FUNCTION_BLOCK "LAxisCtrlApcFr_ChangeModulo"
TITLE = Execute Template
{ S7_Optimized_Access := 'TRUE' }
AUTHOR : SDA
FAMILY : APCFR
VERSION : 1.0
//Template for an FB with Execute / Busy / Done Handling according to PLC Open "Function Blocks for Motion Control"
   VAR_INPUT
      execute { ExternalAccessible := 'False'; ExternalVisible := 'False'; ExternalWritable := 'False'} : Bool;   // Rising edge starts action once
      moduloStartValue { ExternalAccessible := 'False'; ExternalVisible := 'False'; ExternalWritable := 'False'} : LReal;
      moduloLength { ExternalAccessible := 'False'; ExternalVisible := 'False'; ExternalWritable := 'False'} : LReal := 360.0;
      axis { ExternalAccessible := 'False'; ExternalVisible := 'False'; ExternalWritable := 'False'} : DB_ANY;
   END_VAR

   VAR_OUTPUT
      done { ExternalAccessible := 'False'; ExternalVisible := 'False'; ExternalWritable := 'False'} : Bool;   // TRUE: Commanded action has been completed successfully
      busy { ExternalAccessible := 'False'; ExternalVisible := 'False'; ExternalWritable := 'False'} : Bool;   // TRUE: FB is not finished and new output values can be expected
      commandAborted { ExternalAccessible := 'False'; ExternalVisible := 'False'; ExternalWritable := 'False'} : Bool;
      error { ExternalAccessible := 'False'; ExternalVisible := 'False'; ExternalWritable := 'False'} : Bool;   // Rising edge informs that an error occurred during the execution of
      status { ExternalAccessible := 'False'; ExternalVisible := 'False'; ExternalWritable := 'False'} : Word := "STATUS_NO_CALL";   // Current status of FB
      subStatus { ExternalAccessible := 'False'; ExternalVisible := 'False'; ExternalWritable := 'False'} : Word := "ERR_NO_ERROR";
      errorValue { ExternalAccessible := 'False'; ExternalVisible := 'False'; ExternalWritable := 'False'} : Int := 0;
   END_VAR

   VAR
      statExecuteOld { ExternalAccessible := 'False'; ExternalVisible := 'False'; ExternalWritable := 'False'} : Bool;   // Old value of execute for edge detection
      statDone { ExternalAccessible := 'False'; ExternalVisible := 'False'; ExternalWritable := 'False'} : Bool;   // Static value for output done
      statBusy { ExternalAccessible := 'False'; ExternalVisible := 'False'; ExternalWritable := 'False'} : Bool;   // Static value for output busy
      statCommandAborted { ExternalAccessible := 'False'; ExternalVisible := 'False'; ExternalWritable := 'False'} : Bool;
      statError { ExternalAccessible := 'False'; ExternalVisible := 'False'; ExternalWritable := 'False'} : Bool;   // Static value for output error
      statErrorID { ExternalAccessible := 'False'; ExternalVisible := 'False'; ExternalWritable := 'False'} : Word;
      statSubErrorID { ExternalAccessible := 'False'; ExternalVisible := 'False'; ExternalWritable := 'False'} : Word;
      statErrorValue { ExternalAccessible := 'False'; ExternalVisible := 'False'; ExternalWritable := 'False'} : Int;
      statActualStep { ExternalAccessible := 'False'; ExternalVisible := 'False'; ExternalWritable := 'False'} : Int;
      statNextStep { ExternalAccessible := 'False'; ExternalVisible := 'False'; ExternalWritable := 'False'} : Int;
      InstLapcFr_WriteToParameterR_ModuloLength { ExternalAccessible := 'False'; ExternalVisible := 'False'; ExternalWritable := 'False'; S7_SetPoint := 'False'} : "LAxisCtrlApcFr_WriteToParameter";
      InstLapcFr_WriteToParameter_ModuloStartValue { ExternalAccessible := 'False'; ExternalVisible := 'False'; ExternalWritable := 'False'; S7_SetPoint := 'False'} : "LAxisCtrlApcFr_WriteToParameter";
      statStepTimeOut_IN { ExternalAccessible := 'False'; ExternalVisible := 'False'; ExternalWritable := 'False'} : Bool;
      statStepTimeOut_PT { ExternalAccessible := 'False'; ExternalVisible := 'False'; ExternalWritable := 'False'} : Time;
      instStepTimeOut {InstructionName := 'TON_TIME'; LibVersion := '1.0'; ExternalAccessible := 'False'; ExternalVisible := 'False'; ExternalWritable := 'False'; S7_SetPoint := 'False'} : TON_TIME;
   END_VAR

   VAR_TEMP
      tempRefPosAxis {InstructionName := 'TO_PositioningAxis'; LibVersion := '8.0'} : REF_TO TO_PositioningAxis;   // Temporary reference of the technology object type TO_PositioningAxis
   END_VAR


BEGIN
	REGION HEADER
	  //===================================================================================================
	  // SIEMENS SAS    RC-FR DI FA APC
	  //---------------------------------------------------------------------------------------------------
	  // Restrictions:  ---
	  // Requirements:  ---
	  //---------------------------------------------------------------------------------------------------
	  // Description:   Changing modulo value of axis
	  //---------------------------------------------------------------------------------------------------
	  // Change log table:
	  // Version  Date        TIA   Expert  Changes applied
	  // 01.00    2020.07.24  V16   SDA     First released version
	  // 01.01    2021.06.01  V16   SDA     Name changed
	  // 01.02    2022.04.20  V17   FGe     Bugfix: incorrect error value step 40
	  //                                    Moved constants TO global definition
	  // 05.00    2024.09.11  V19   SDa     Adaptation with DBAny type #axis
	  //---------------------------------------------------------------------------------------------------
	  // Compatibility to TIA version require the use of latest version for PLC fimware and Motion Control
	  // e.g; Firmware 3.1 and Motion Control V8.0 for TIA V19
	  //===========================================================================================
	END_REGION

	REGION INITIALISATION
	    #tempRefPosAxis ?= #axis;
	END_REGION

	IF (#tempRefPosAxis <> NULL) THEN
	    // Axis type is TO_PositioningAxis or TO_SynchronousAxis

	    REGION INSTANCES
	        //------------------------------------------------------------------------------------------
	        // TODO: Insert here instances of MC instructions.
	        // inputs / outputs to be set / used in main section

	        #instStepTimeOut(IN := #statStepTimeOut_IN,
	                         PT := #statStepTimeOut_PT);

	        #InstLapcFr_WriteToParameterR_ModuloLength("TO" := #tempRefPosAxis^,
	                                                   restart := false,
	                                                   parameterValue := #moduloLength,
	                                                   TO_Parameter := #tempRefPosAxis^.Modulo.Length);

	        #InstLapcFr_WriteToParameter_ModuloStartValue("TO" := #tempRefPosAxis^,
	                                                      restart := true,
	                                                      parameterValue := #moduloStartValue,
	                                                      TO_Parameter := #tempRefPosAxis^.Modulo.StartValue);
	        //-----------------------------------------------------------------------------------
	    END_REGION

	    REGION CALL HANDLING

	        //Check if FB is triggered
	        IF #execute AND NOT #statExecuteOld
	            // if FB should finish current job before new job can be started with rising edge of execute,
	            // you must remove the first comment character on next line
	            AND NOT #statBusy
	        THEN
	            REGION FB TRIG (FIRST CALL)
	                //-----------------------------------------------------------------------------------
	                //TODO: Initialize functionality after triggering FB, e.g. reset of values
	                //
	                // Timers
	                #statStepTimeOut_IN := FALSE;
	                // Commands
	                #InstLapcFr_WriteToParameterR_ModuloLength.write := FALSE;
	                #InstLapcFr_WriteToParameter_ModuloStartValue.write := FALSE;
	                // Status
	                #statNextStep := 10;
	                #statErrorID := "STATUS_FIRST_CALL";
	                #statSubErrorID := "ERR_NO_ERROR";
	                //-----------------------------------------------------------------------------------

	                //Functionality is busy
	                #statDone := FALSE;
	                #statBusy := TRUE;
	                #statCommandAborted := FALSE;
	                //Reset diagnostic
	                #statError := FALSE;
	                #statErrorID := "ERR_NO_ERROR";
	                #statSubErrorID := "ERR_NO_ERROR";
	                #statErrorValue := 0;
	                // Write outputs
	                #done := #statDone;
	                #busy := #statBusy;
	                #commandAborted := #statCommandAborted;
	                #error := #statError;
	                #status := "STATUS_FIRST_CALL";
	                #subStatus := #statSubErrorID;
	                #errorValue := #statErrorValue;
	                #statExecuteOld := #execute;
	                RETURN;
	            END_REGION

	            //FB is currently inactive
	        ELSIF NOT #execute AND NOT #statBusy AND NOT #statExecuteOld
	        THEN
	            REGION NO CALL
	                //Outputs are reset with falling edge of enable input
	                //Write outputs
	                #done := #statDone;
	                #busy := #statBusy;
	                #commandAborted := #statCommandAborted;
	                #error := #statError;
	                #status := "STATUS_NO_CALL";
	                #subStatus := "ERR_NO_ERROR";
	                #errorValue := 0;
	                #statExecuteOld := #execute;
	                RETURN;
	            END_REGION

	            //FB is currently executed and not finished
	        ELSIF #statBusy OR #execute
	        THEN
	            REGION BUSY
	                #statExecuteOld := #execute OR #statBusy;
	            END_REGION

	            //FB finished job
	        ELSE
	            REGION LAST CALL
	                //-----------------------------------------------------------------------------------
	                //TODO: Initialize functionality after triggering FB, e.g. reset of values
	                //
	                // Timers
	                #statStepTimeOut_IN := FALSE;
	                // Commands
	                #InstLapcFr_WriteToParameterR_ModuloLength.write := FALSE;
	                #InstLapcFr_WriteToParameter_ModuloStartValue.write := FALSE;
	                // State
	                #statNextStep := 0;
	                //-----------------------------------------------------------------------------------
	                #statDone := FALSE;
	                #statBusy := FALSE;
	                #statCommandAborted := FALSE;
	                #statError := FALSE;
	                #statErrorID := "ERR_NO_ERROR";
	                #statSubErrorID := "ERR_NO_ERROR";
	                #statErrorValue := 0;
	                #statExecuteOld := #execute;
	                RETURN;
	            END_REGION

	        END_IF;
	    END_REGION ;

	    REGION USER PROGRAM
	        //-----------------------------------------------------------------------------------
	        //TODO: Add user program
	        //
	        //Following values have to be set in user program:
	        //  - statDone:     FB is finished with execution
	        //  - statAborted   Execution is aborted by an external command
	        //  - statError:    Error happened in program
	        //  - statStatus:   Identifier for current error
	        //  - statSubStatus:Identifier for subcall error
	        //
	        //Following values are not allowed to use in user program:
	        //  - statBusy
	        //  - status, subStatus, aborted, busy, done and error
	        //
	        //Attention:
	        //  - Input parameters can be updated continously
	        //  - If inputs exceed application limits, system has either to throw an error or to correct it
	        //      automatically
	        //-----------------------------------------------------------------------------------

	        REGION CHANGE MODULO VALUES

	            // update running step
	            #statActualStep := #statNextStep;
	            CASE #statActualStep OF

	                10: // Init values
	                    REGION INITIALISATION
	                        // Next step
	                        #statNextStep := 20;
	                    END_REGION

	                20: // Check change modulo conditions
	                    REGION CHECK CONDITIONS
	                        IF NOT #tempRefPosAxis^.Modulo.Enable THEN
	                            // module not activated
	                            #statErrorID := "ERR_CM_MODULO_NOT_ACTIVATED";
	                            #statNextStep := 900;

	                        ELSIF #moduloLength <= 0 THEN
	                            // wrong length
	                            #statErrorID := "ERR_CM_LENGTH_VALUE";
	                            #statNextStep := 900;

	                        ELSIF #tempRefPosAxis^.StatusWord.%X0 THEN
	                            // axis enabled
	                            #statErrorID := "ERR_CM_AXIS_ENABLED";
	                            #statNextStep := 900;

	                        ELSE
	                            // Next step
	                            #statNextStep := 30;
	                        END_IF;
	                    END_REGION

	                30: // change length value
	                    REGION CHANGE MODULO LENGTH VALUE
	                        // Step timeout
	                        #statStepTimeOut_PT := "LAPCFR_CM_WRITE_TOPARAMETER_TIMEOUT";
	                        #statStepTimeOut_IN := true;

	                        #InstLapcFr_WriteToParameterR_ModuloLength.write := TRUE;

	                        IF #InstLapcFr_WriteToParameterR_ModuloLength.error THEN
	                            #statErrorID := "ERR_CM_WRITEPARAMETER_LENGTHVALUE";
	                            #statSubErrorID := #InstLapcFr_WriteToParameterR_ModuloLength.status;
	                            #InstLapcFr_WriteToParameterR_ModuloLength.write := FALSE;
	                            #statStepTimeOut_IN := FALSE;
	                            #statNextStep := 900;

	                        ELSIF #InstLapcFr_WriteToParameterR_ModuloLength.done THEN
	                            #InstLapcFr_WriteToParameterR_ModuloLength.write := FALSE;
	                            #statStepTimeOut_IN := FALSE;
	                            // Next step
	                            #statNextStep := 40;

	                        ELSIF #instStepTimeOut.Q THEN
	                            // write parameter timeout
	                            #statErrorID := "ERR_CM_WRITEPARAMETER_TIMEOUT_LENGTHVALUE";
	                            #InstLapcFr_WriteToParameterR_ModuloLength.write := FALSE;
	                            #statStepTimeOut_IN := FALSE;
	                            #statNextStep := 900;
	                        END_IF;

	                    END_REGION

	                40: // change start value
	                    REGION CHANGE MODULO START VALUE
	                        // Step timeout
	                        #statStepTimeOut_PT := "LAPCFR_CM_WRITE_TOPARAMETER_TIMEOUT";
	                        #statStepTimeOut_IN := true;

	                        #InstLapcFr_WriteToParameter_ModuloStartValue.write := TRUE;

	                        IF #InstLapcFr_WriteToParameter_ModuloStartValue.error THEN
	                            #statErrorID := "ERR_CM_WRITEPARAMETER_STARTVALUE";
	                            #statSubErrorID := #InstLapcFr_WriteToParameter_ModuloStartValue.status;
	                            #InstLapcFr_WriteToParameter_ModuloStartValue.write := FALSE;
	                            #statStepTimeOut_IN := FALSE;
	                            #statNextStep := 900;

	                        ELSIF #InstLapcFr_WriteToParameter_ModuloStartValue.done THEN
	                            #InstLapcFr_WriteToParameter_ModuloStartValue.write := FALSE;
	                            #statStepTimeOut_IN := FALSE;
	                            // Next step
	                            #statNextStep := 120;

	                        ELSIF #instStepTimeOut.Q THEN
	                            // write parameter timeout
	                            #statErrorID := "ERR_CM_WRITEPARAMETER_TIMEOUT_STARTVALUE";
	                            #InstLapcFr_WriteToParameterR_ModuloLength.write := FALSE;
	                            #InstLapcFr_WriteToParameter_ModuloStartValue.write := FALSE;
	                            #statStepTimeOut_IN := FALSE;
	                            #statNextStep := 900;
	                        END_IF;

	                    END_REGION

	                120://Function Ok
	                    REGION FUNCTION_DONE
	                        #statDone := TRUE;
	                    END_REGION ;

	                900:  //Fault handling
	                    REGION FUNCTION_FAULTY
	                        #statNextStep := 910;
	                    END_REGION

	                910:   // change modulo values ended with fault
	                    #statError := TRUE;

	            END_CASE;

	            IF #statNextStep = 900 AND #statActualStep <> 900 THEN
	                // Store faulty step
	                #statErrorValue := #statActualStep;
	            END_IF;

	        END_REGION

	        //
	        //-----------------------------------------------------------------------------------
	    END_REGION

	    REGION ERROR_HANDLING

	        //Error occured in request
	        IF #statError
	        THEN
	            #statDone := FALSE;
	            #statCommandAborted := FALSE;
	            #statBusy := FALSE;
	            //-----------------------------------------------------------------------------------
	            //TODO: Set correct status that identifies error clearly if not set in user program region
	            // #statStatus := ...;
	            // #statSubStatus := ...;
	            //
	            #status := #statErrorID;
	            #subStatus := #statSubErrorID;
	            #errorValue := #statErrorValue;
	            //-----------------------------------------------------------------------------------

	            // Resquest aborted
	        ELSIF #statCommandAborted
	        THEN
	            #statDone := FALSE;
	            #statBusy := FALSE;
	            #statError := FALSE;
	            #status := "STATUS_EXECUTION_ABORTED";
	            #subStatus := "ERR_NO_ERROR";
	            #errorValue := 0;

	            //Request finished
	        ELSIF #statDone
	        THEN
	            #statBusy := FALSE;
	            #statCommandAborted := FALSE;
	            #statError := FALSE;
	            #status := "STATUS_FINISHED_NOERROR";
	            #subStatus := "ERR_NO_ERROR";
	            #errorValue := 0;

	            //Request in execution
	        ELSE
	            #status := "STATUS_SUBSEQUENT_CALL";
	            #subStatus := "ERR_NO_ERROR";
	            #errorValue := 0;
	        END_IF;

	        //Write static values to outputs
	        #done := #statDone;
	        #busy := #statBusy;
	        #commandAborted := #statCommandAborted;
	        #error := #statError;
	    END_REGION
	    //-----------------------------------------------------------------------------------

	ELSE
	    IF #execute THEN
	        // Invalid TO specification
	        #error := TRUE;
	        #done := FALSE;
	        #busy := FALSE;
	        #status := "ERROR_INVALID_TECHNOLOGY_OBJECT"; // Invalid TO specification
	        #subStatus := "ERR_NO_ERROR";
	    ELSE
	        #error := FALSE;
	        #done := FALSE;
	        #busy := FALSE;
	        #status := "ERR_NO_ERROR";
	        #subStatus := "ERR_NO_ERROR";
	    END_IF;
	END_IF;
END_FUNCTION_BLOCK

